// TIA Portal V15 export
// export: Created 2019-02-06T17:41:42.9000068Z, ExportSetting WithDefaults, WithReadOnly, DisplayName Totally Integrated Automation Portal, DisplayVersion V15 Update 2, DisplayName TIA Portal Openness, DisplayVersion V15 Update 2, DisplayName STEP 7 Professional, DisplayVersion V15 Update 2, DisplayName STEP 7 Safety, DisplayVersion V15, DisplayName WinCC Professional, DisplayVersion V15 Update 2, DisplayName SIMATIC Visualization Architect, DisplayVersion V15 Update 1
TYPE "iUDT_PO_ADRxx34_APPL_ROBNAME"
// stored: CreationDate 2016-06-13T08:33:18.8280064Z, InterfaceModifiedDate 2017-05-29T07:30:56.8116619Z, IsConsistent true, IsKnowHowProtected false, LibraryConformanceStatus The object is library-conformant., ModifiedDate 2018-01-29T16:41:47.0308707Z
   STRUCT
      "RB-PLC" : Struct   // RB-PLC interlocks
      END_STRUCT;
      "RB-RB" : Struct   // RB-RB interlock signal
      END_STRUCT;
   END_STRUCT;
END_TYPE
